ABB RobotStudio station: SmartComponentSolution.rspag

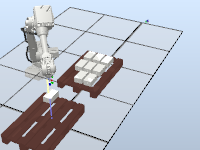
--- station ---
Station SmartComponentSolution (saved by RobotStudio 20.2.9116.0)
Controller IRB_4600_60kg_2.05m, task T_ROB1: task frame (RAPID world) sits at (1429.89, 1152.71, -186.83) mm in the station
Controller IRB_4600_60kg_2.05m
  mechanical unit ROB_1: IRB4600_60_205_C_01, 6 joints, base frame (0, 0, 0) mm
Layout (positions relative to the parent item):
  - IRB4600_60_205_C_01 [mechanism, from Robots\IRB4600_60_205_C_G_01.rslib] at (1429.89, 1152.71, -186.83) mm; joint values [-2.43, 0.3631, 0.2506, 0, 0.9571, 0.7116] (rad or m)
  - Connector [part] at (2207.99, -409.6, 387.37) mm, rotated rx 90 ry 0 rz 0 deg
  - OD1-B100H50I14-S098974 [part] at (3104.69, -456.71, 431.38) mm, rotated rx 0 ry 90 rz -90 deg
  - Box [part] at (384.63, 251.78, 140.86) mm, rotated rx 90 ry 0 rz 0 deg
  - Euro Pallet [graphiccomponentgroup, from Equipment\Euro Pallet.rslib] at (680.82, -151.09, 0) mm
    - Body 1 [part, from Equipment\Euro Pallet.rslib] at (188.03, -194.52, 0) mm
  - SC_VaccumGripperDetector [smart component] at (384.55, 251.34, 604.68) mm, rotated rx 180 ry 0 rz 0 deg
      signals: DO sensorSignal, DI Attached, DI Detach
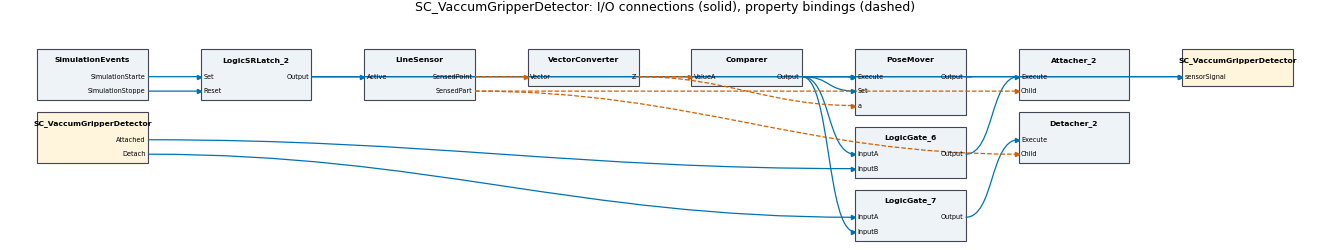
      connections:
        SimulationEvents.SimulationStarted -> LogicSRLatch_2.Set
        SimulationEvents.SimulationStopped -> LogicSRLatch_2.Reset
        LogicSRLatch_2.Output -> LineSensor.Active
        LogicSRLatch_2.Output -> PoseMover.Execute
        LogicSRLatch_2.Output -> Positioner.Execute
        Comparer.Output -> LogicSRLatch_6.Set
        LogicSRLatch_6.Output -> PoseMover_3.Execute
        LogicSRLatch_6.Output -> SC_VaccumGripperDetector.sensorSignal
        Comparer.Output -> SC_VaccumGripperDetector.sensorSignal
        Comparer.Output -> LogicGate_6.InputA
        SC_VaccumGripperDetector.Attached -> LogicGate_6.InputB
        LogicGate_6.Output -> Attacher_2.Execute
        SC_VaccumGripperDetector.Detach -> LogicGate_7.InputA
        Comparer.Output -> LogicGate_7.InputB
        LogicGate_7.Output -> Detacher_2.Execute
        LineSensor.SensedPoint => VectorConverter.Vector
        VectorConverter.Z => Comparer.ValueA
        VectorConverter.Z => Expression.a
        LineSensor.SensedPart => Attacher_2.Child
        LineSensor.SensedPart => Detacher_2.Child
    - small_suction_gripper_2 [mechanism] at (0, 0, 0.06) mm
        TCP small_suction_gripper at (-62.96, -41.92, 61.7) mm, rotated rx 90 ry 0 rz 0 deg
        links: suction gripper-2_3
    - LineSensor [smart component, from Components\LineSensor.rslib] at (-638.5, 408.61, -364.87) mm
        properties: Start=[0.641250538776752 -0.457606 0.455378]; End=[0.641250538776752 -0.457606 1.042378]; Radius=0.001; SensedPart=Box; SensedPoint=[0.387301147460938 0.300343078613281 0.241100891113281]
      - _sensorPart_ [part]
    - Comparer [smart component, from Components\Comparer.rslib]
        properties: ValueA=0.241100891113281; Operator=>; ValueB=0.2
    - VectorConverter [smart component, from Components\VectorConverter.rslib]
        properties: X=0.387301147460938; Y=0.300343078613281; Z=0.241100891113281; Vector=[0.387301147460938 0.300343078613281 0.241100891113281]
    - SimulationEvents [smart component, from Components\SimulationEvents.rslib]
    - LogicSRLatch_2 [smart component, from Components\LogicSRLatch.rslib]
    - Attacher_2 [smart component, from Components\Attacher.rslib]
        properties: Parent=small_suction_gripper_2; Flange=0; Child=Box; Mount=false; Offset=[0 0 0]; Orientation=[0 0 0]
    - LogicGate_6 [smart component, from Components\LogicGate.rslib]
        properties: Operator=AND; Delay=0
    - Detacher_2 [smart component, from Components\Detacher.rslib]
        properties: Child=Box; KeepPosition=true
    - LogicGate_7 [smart component, from Components\LogicGate.rslib]
        properties: Operator=AND; Delay=0
  - OD1-B100H50I14-S098974_2 [part] at (319.44, 299.44, 538.17) mm, rotated rx -126.79 ry -90 rz 36.79 deg
  - Connector_2 [part] at (376.89, 260.94, 582.18) mm, rotated rx -90 ry 0 rz 0 deg
  - Box_2 [part] at (1100.5, 65.48, 144.74) mm, rotated rx 90 ry 0 rz 0 deg
  - Box_3 [part] at (1100.5, -122.34, 144.74) mm, rotated rx 90 ry 0 rz 0 deg
  - Box_4 [part] at (1445.39, 246.78, 144.74) mm, rotated rx 90 ry 0 rz 0 deg
  - Box_5 [part] at (1444.74, 62.09, 144.74) mm, rotated rx 90 ry 0 rz 0 deg
  - Box_6 [part] at (1450.77, -121.77, 144.74) mm, rotated rx 90 ry 0 rz 0 deg
  - Box_7 [part] at (1788.47, 246.78, 144.74) mm, rotated rx 90 ry 0 rz 0 deg
  - Box_8 [part] at (1789.72, 54.43, 144.74) mm, rotated rx 90 ry 0 rz 0 deg
  - Box_9 [part] at (1780.97, -127.61, 144.74) mm, rotated rx 90 ry 0 rz 0 deg
  - Euro Pallet_2 [graphiccomponentgroup, from Equipment\Euro Pallet.rslib] at (-902.1, -151.09, 0) mm
    - Body 1 [part, from Equipment\Euro Pallet.rslib] at (188.03, -194.52, 0) mm
  - LogicSRLatch_7 [smart component, from Components\LogicSRLatch.rslib]
  - LogicGate_4 [smart component, from Components\LogicGate.rslib]
      properties: Operator=NOT; Delay=0
  - Frame_1 [frame] at (3169.8, -408.61, 483.89) mm
Attachment: OD1-B100H50I14-S098974_2 is attached to DEFAULT-34
Attachment: Connector_2 is attached to DEFAULT-34
Attachment: SC_VaccumGripperDetector is attached to IRB4600_60_205_C_01 / Link6
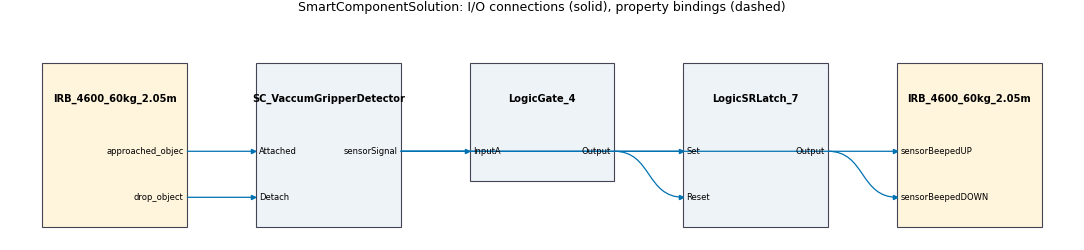
Station logic (signal -> signal, property => property):
  SC_VaccumGripperDetector.sensorSignal -> IRB_4600_60kg_2.05m.sensorBeepedUP
  SC_VaccumGripperDetector.sensorSignal -> LogicSRLatch_7.Set
  SC_VaccumGripperDetector.sensorSignal -> LogicGate_4.InputA
  LogicGate_4.Output -> LogicSRLatch_7.Reset
  LogicSRLatch_7.Output -> IRB_4600_60kg_2.05m.sensorBeepedDOWN
  IRB_4600_60kg_2.05m.approached_object -> SC_VaccumGripperDetector.Attached
  IRB_4600_60kg_2.05m.drop_object -> SC_VaccumGripperDetector.Detach

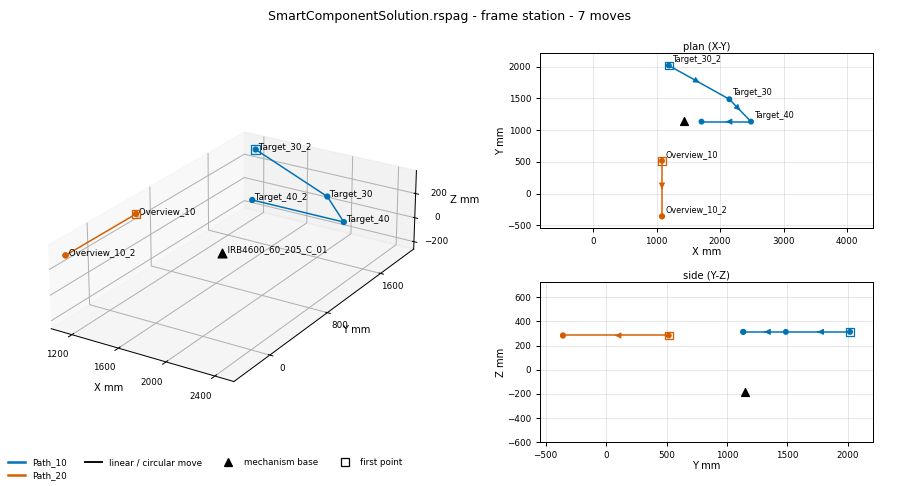
[picture p0: tool path of SmartComponentSolution.rspag in frame station, 7 of 18 moves have a stored position in this frame; points joined in program order, loops and branches not executed]
--- Backups/IRB_4600_60kg_2.05m/RAPID/TASK1/PROGMOD/CalibData.mod ---
MODULE CalibData
    PERS tooldata small_suction_gripper:=[TRUE,[[-0.000055309,0.000726868,121.499905969],[1,0.000000005,0.000000013,-0.000000029]],[1,[0.443001337,-9.457000743,69.908999891],[1,0,0,0],0,0,0]];
ENDMODULE

--- Backups/IRB_4600_60kg_2.05m/RAPID/TASK1/PROGMOD/Module1.mod ---
MODULE Module1
    CONST robtarget Target_30_2:=[[-237.219768702,866.283675835,500],[0,1,0,0],[0,0,-2,0],[9E+09,9E+09,9E+09,9E+09,9E+09,9E+09]];
    CONST robtarget Target_30:=[[716.121686162,335.077687596,500],[0,1,0,0],[0,0,-2,0],[9E+09,9E+09,9E+09,9E+09,9E+09,9E+09]];
    CONST robtarget Target_40:=[[1057.065915871,-17.60100368,500],[0,1,0,0],[0,-1,-2,0],[9E+09,9E+09,9E+09,9E+09,9E+09,9E+09]];
    CONST robtarget Target_40_2:=[[277.117965124,-17.60100368,500],[0,1,0,0],[0,0,-2,0],[9E+09,9E+09,9E+09,9E+09,9E+09,9E+09]];
    CONST robtarget Overview_10:=[[-345.337592383,-634.2218361,470],[0,1,0,0],[0,0,0,0],[9E+09,9E+09,9E+09,9E+09,9E+09,9E+09]];
    CONST robtarget Overview_10_2:=[[-345.337592383,-1509.837410954,470],[0,1,0,0],[0,0,0,0],[9E+09,9E+09,9E+09,9E+09,9E+09,9E+09]];
    CONST robtarget Overview_10_3:=[[12.284555899,-1493.428131522,431.52658222],[0,1,0,0],[0,0,0,0],[9E+09,9E+09,9E+09,9E+09,9E+09,9E+09]];
    CONST robtarget Overview_10_4:=[[11.425088297,-611.443739064,431.52658222],[0,1,0,0],[0,0,0,0],[9E+09,9E+09,9E+09,9E+09,9E+09,9E+09]];
    CONST robtarget Overview_10_5:=[[353.203433771,-634.2218361,431.52658222],[0,1,0,0],[0,0,0,0],[9E+09,9E+09,9E+09,9E+09,9E+09,9E+09]];
    CONST robtarget Overview_10_6:=[[379.156403723,-1514.983024916,431.52658222],[0,1,0,0],[0,0,0,0],[9E+09,9E+09,9E+09,9E+09,9E+09,9E+09]];
    CONST num x_vacuum_offset := 1097.85-1100.6;
    CONST num y_vacuum_offset := 197.02-246.02;


    VAR robtarget p4;
    VAR robtarget p5;
    VAR robtarget p6;
    VAR robtarget p7;

    VAR robtarget p8;
    VAR robtarget p9;
    VAR robtarget p10;
    VAR robtarget p11;
    VAR robtarget p12;
    VAR robtarget p13;
    VAR robtarget p14;

    VAR pose frame1;

!***********************************************************
    !
    ! Module:  Module1
    !
    ! Description:
    !   <Insert description here>
    !
    ! Author: jelac
    !
    ! Version: 1.0
    !
    !***********************************************************


    !***********************************************************
    !
    ! Procedure main
    !
    !   This is the entry point of your program
    !
    !***********************************************************
    PROC main()
        !Add your code here
        Path_20;
    ENDPROC
    PROC Path_10()
        MoveL Target_30_2,v1000,z100,small_suction_gripper\WObj:=wobj0;
        MoveL Target_30,v1000,z100,small_suction_gripper\WObj:=wobj0;
        MoveL Target_40,v1000,z100,small_suction_gripper\WObj:=wobj0;
        MoveL Target_40_2,v1000,z100,small_suction_gripper\WObj:=wobj0;
    ENDPROC
    PROC Path_20()

        Reset approached_object;
        Set drop_object;

        MoveL Overview_10,v300,z100,small_suction_gripper\WObj:=wobj0;
        SearchL \Stop, sensorBeepedUP, p4, Overview_10_2, v50, small_suction_gripper\WObj:=wobj0;
        p5 := p4;
        p5.trans.y := p5.trans.y-50;
        !p5.trans.z := p5.trans.z+100;
        p12 := p5;
        MoveL p5,v300,z100,small_suction_gripper\WObj:=wobj0;
        p7 := p5;
        p7.trans.x := p5.trans.x-300;

        SearchL \Stop,  sensorBeepedUP,\NegFlank, p6, p7, v50, small_suction_gripper\WObj:=wobj0;
        MoveL p5,v300,z100,small_suction_gripper\WObj:=wobj0;
        SearchL \Stop,  sensorBeepedUP,\NegFlank, p8, Overview_10_2, v50, small_suction_gripper\WObj:=wobj0;
        p10 := p5;
        p10.trans.x := p10.trans.x + 400;
        MoveL p5,v300,z100,small_suction_gripper\WObj:=wobj0;
        SearchL \Stop,  sensorBeepedUP,\NegFlank, p9, p10, v50, small_suction_gripper\WObj:=wobj0;

        p11 := p5;
        p11.trans.y := (p4.trans.y+p8.trans.y)/2 - y_vacuum_offset;
        p11.trans.x := (p6.trans.x+p9.trans.x)/2 - x_vacuum_offset;

        MoveL p11,v80,z100,small_suction_gripper\WObj:=wobj0;

        p11.trans.z := p11.trans.z - 38;
        MoveL p11,v300,z100,small_suction_gripper\WObj:=wobj0;

        WaitTime(5);
        Reset drop_object;
        Set approached_object;
        p12.trans.z := p12.trans.z+200;
        MoveL p12,v300,z100,small_suction_gripper\WObj:=wobj0;
        p13 := p12;
        p13.trans.x := p13.trans.x - 700;
        MoveL p13,v300,z100,small_suction_gripper\WObj:=wobj0;
        p14 := p13;
        p14.trans.z := p13.trans.z - 240.94;
        MoveL p14,v300,z100,small_suction_gripper\WObj:=wobj0;
        WaitTime(5);
        Reset approached_object;
        Set drop_object;

        MoveL p13,v300,z100,small_suction_gripper\WObj:=wobj0;

    ENDPROC
    PROC Seek_box()


    ENDPROC
ENDMODULE

--- Backups/IRB_4600_60kg_2.05m/SYSPAR/EIO.cfg ---
EIO:CFG_1.0:6:1::
#
EIO_SIGNAL:

      -Name "pointFound" -SignalType "DO" -Access "All"

      -Name "sensorBeepedUP" -SignalType "DI" -Access "All"

      -Name "sensorBeepedDOWN" -SignalType "DI" -Access "All"

      -Name "approached_object" -SignalType "DO" -Access "All"

      -Name "drop_object" -SignalType "DO" -Access "All"
